// TIA Portal V20 export
DATA_BLOCK "BK29"   // DB280
// stored: MemoryReserve 100
   VAR
      "X10-1.SUCTION PAD TOP LEFT VACUUM ON" : Bool := FALSE;
      "X10-2.SUCTION PAD TOP LEFT VACUUM OFF" : Bool := FALSE;
      "X12-1.SUCTION PAD TOP RIGHT VACUUM ON" : Bool := FALSE;
      "X12-2.SUCTION PAD TOP RIGHT VACUUM OFF" : Bool := FALSE;
      "X14-1.SUCTION PAD BTM LEFT VACUUM ON" : Bool := FALSE;
      "X14-2.SUCTION PAD BTM LEFT VACUUM OFF" : Bool := FALSE;
      "X16-1.SUCTION PAD BTM RIGHT VACUUM ON" : Bool := FALSE;
      "X16-2.SUCTION PAD BTM RIGHT VACUUM OFF" : Bool := FALSE;
   END_VAR
BEGIN
END_DATA_BLOCK
